// Block: A0303_Manager_PERS

DATA_BLOCK A0303_Manager_PERS
VERSION : 0.1
   NON_RETAIN
   VAR
      Par : Struct
         Antiribaltamento : Struct
            Offset_Pos : LReal;
         END_STRUCT;
      END_STRUCT;
   END_VAR

BEGIN
   // No initialization required
END_DATA_BLOCK
